Staubli VAL3: HIT_YD.pjx

--- HIT_YD.pjx ---
Parameters version=s7.6.4 stackSize=5000 millimeterUnit=true
Program file=blow.pgx
Program file=bypassPick.pgx
Program file=cellManager.pgx
Program file=getToolStatus.pgx
Program file=goHome.pgx
Program file=init.pgx
Program file=initTracking.pgx
Program file=isInSafetyArea.pgx
Program file=ModbusGet.pgx
Program file=modbusSet.pgx
Program file=OMAC_Abort.pgx
Program file=OMAC_Hold.pgx
Program file=OMAC_Main.pgx
Program file=OMAC_Reset.pgx
Program file=OMAC_Start.pgx
Program file=OMAC_Stop.pgx
Program file=OMAC_Unhold.pgx
Program file=overflowPick.pgx
Program file=Place.pgx
Program file=productionCycle.pgx
Program file=robot2PC.pgx
Program file=robot2PLC.pgx
Program file=send2NextRob.pgx
Program file=setAlarm.pgx
Program file=setConvSpeed.pgx
Program file=start.pgx
Program file=stop.pgx
Program file=trackErr_init.pgx
Program file=trackingPick.pgx
Program file=transferQueue.pgx
Data file=HIT_YD.dtx
Library alias=mot path=Disk://Tracking/Motion/Motion.pjx
Type name=object path=Disk://Tracking/Templates/object/object.pjx

--- HIT_YD.dtx ---
aio aConvSpeed = {link=ModbusSrv-0\Modbus-Word\ao[3]}
aio aPlcCmd = {link=ModbusSrv-0\Modbus-Word\ai[0]}
aio aRbAlarm = {link=ModbusSrv-0\Modbus-Word\ao[0]}
aio aRbStatus = {link=ModbusSrv-0\Modbus-Word\ao[1]}
bool _bConvExist = true
bool _bEndCycle
bool _bIsPicking
bool _bIsPlacing
bool _bMutexCnvQueue
bool _bOverflowed = true
bool _bPartInTool = true
bool _bSentToHome
bool _bVisionOK = true
bool bLockPage
bool bPickDetection
bool bSetConvSpeed
bool bSyn
bool bTransferData = true
dio dAlarm[8]
  [0] = {link=ModbusSrv-0\Modbus-Bit\do[8]}
  [1] = {link=ModbusSrv-0\Modbus-Bit\do[9]}
  [2] = {link=ModbusSrv-0\Modbus-Bit\do[10]}
  [3] = {link=ModbusSrv-0\Modbus-Bit\do[11]}
  [4] = {link=ModbusSrv-0\Modbus-Bit\do[12]}
  [5] = {link=ModbusSrv-0\Modbus-Bit\do[13]}
  [6] = {link=ModbusSrv-0\Modbus-Bit\do[14]}
  [7] = {link=ModbusSrv-0\Modbus-Bit\do[15]}
dio dBlow = {link=BasicIO-1\%Q5}
dio dConvControl[2]
  [0] = {link=BasicIO-1\%I4}
  [1] = {link=BasicIO-1\%Q6}
dio dPartInTool = {link=fIn0}
dio dPermitPlace[4]
  [0] = {link=BasicIO-1\%I3}
  [1] = {link=BasicIO-1\%I2}
  [2] = {link=BasicIO-1\%I1}
  [3] = {link=BasicIO-1\%I0}
dio dPlaceDone[4]
  [0] = {link=BasicIO-1\%Q11}
  [1] = {link=BasicIO-1\%Q10}
  [2] = {link=BasicIO-1\%Q9}
  [3] = {link=BasicIO-1\%Q8}
dio dStartControl[4]
  [0] = {link=ModbusSrv-0\Modbus-Bit\di[4]}
  [1] = {link=ModbusSrv-0\Modbus-Bit\di[5]}
  [2] = {link=ModbusSrv-0\Modbus-Bit\di[6]}
  [3] = {link=ModbusSrv-0\Modbus-Bit\di[7]}
dio dStartState[4]
  [0] = {link=ModbusSrv-0\Modbus-Bit\do[4]}
  [1] = {link=ModbusSrv-0\Modbus-Bit\do[5]}
  [2] = {link=ModbusSrv-0\Modbus-Bit\do[6]}
  [3] = {link=ModbusSrv-0\Modbus-Bit\do[7]}
dio dVacuum = {link=BasicIO-1\%Q4}
frame fConveyor = {x=365.904087, y=326.91934, z=-82.602337, rx=-0.010861, ry=-0.059106, rz=0.004608, fatherId=world[0]}
frame fDetection = {x=392.598601, y=461.346273, z=-82.976862, rx=0.205045, ry=0.617271, rz=0.011036, fatherId=world[0]}
jointRs jDropPart = {j1=102.785955, j2=-95.43121, j3=69.578977, j4=134.260732}
jointRs jHome = {j1=102.785955, j2=-95.43121, j3=69.578977, j4=134.260732}
jointRs jPark = {j1=102.785955, j2=-95.43121, j3=69.578977, j4=134.260732}
mdesc _mLoad = {accel=133.4025, vel=115.5, decel=133.4025}
mdesc mLoad = {accel=121, vel=110, decel=121}
mdesc mNomSpeed = {accel=144, vel=120, decel=144, leave=20, reach=20}
mdesc mPickDown = {accel=144, vel=120, decel=144, leave=10, reach=10, blend=off}
mdesc mPickup = {accel=121, vel=110, decel=121, leave=40, reach=40}
mdesc mPlaceDown = {accel=144, vel=120, decel=144, leave=15, reach=15, blend=off}
mdesc mPlaceUp = {accel=144, vel=120, decel=144, leave=20, reach=20, blend=cartesian}
mdesc mSlow = {accel=1, vel=10, decel=1, leave=10, reach=10}
mdesc mUnload = {accel=144, vel=120, decel=144, leave=40, reach=40}
num _nBlowDelay
num _nCntBypassed = 1
num _nCntPartsDone[2]
  [0] = 74956
  [1] = 74907
num _nCntTransfered = 8
num _nConvSpd
num _nCycleTime[4]
  [0] = 33.16
  [1] = 2.331
  [2] = 48.87
  [3] = 0.935
num _nCycleTimeIndx
num _nID = -1
num _nLastStateCMD
num _nOmacStat = 3
num _nPartID = 1
num _nPlaceCurItem[2]
num _nPullIndexTQ = 8
num _nPushIndexTQ = 8
num _nStateCMD
num _nTimer = 355.546
num _nTrackErr = 315
num nBlowID = 0.3
num nBypass = 1
num nLoadRatio[4]
  [0] = 0.7
  [1] = 0.85
  [2] = 0.95
  [3] = 1.05
num nNomConvSpeed = 100
num nPartHeight = 6
num nPickAppro = 65
num nPickOS_X = -3
num nPickOS_Y
num nPlaceAppro = 60
public num nPlaceNum = 3
num nSafeMaxX = 850
num nSafeMaxY = 650
num nSafeMinX
num nSafeMinY
num nStopTime = 0.02
num nTestData[5]
  [0] = 6
  [1] = -49
  [2] = 55
  [4] = 24206
num nVacuumID
num nWaitDist2Up4BP = -300
num nWaitDistToDown = 50
num nWaitDistToUp[1 3]
  [0,0] = -80
  [0,1] = 120
  [0,2] = 400
num nWaitDistX
object _oTransferQueue[1 100]
  [0,0]
    num nID = -1
    num nLatchedValue
    trsf trTrsf
  [0,1]
    num nID = -1
    num nLatchedValue
    trsf trTrsf
  [0,2]
    num nID = -1
    num nLatchedValue
    trsf trTrsf
  [0,3]
    num nID = -1
    num nLatchedValue
    trsf trTrsf
  [0,4]
    num nID = -1
    num nLatchedValue
    trsf trTrsf
  [0,5]
    num nID = -1
    num nLatchedValue
    trsf trTrsf
  [0,6]
    num nID = -1
    num nLatchedValue
    trsf trTrsf
  [0,7]
    num nID = -1
    num nLatchedValue
    trsf trTrsf
  [0,8]
    num nID = -1
    num nLatchedValue
    trsf trTrsf
  [0,9]
    num nID = -1
    num nLatchedValue
    trsf trTrsf
  [0,10]
    num nID = -1
    num nLatchedValue
    trsf trTrsf
  [0,11]
    num nID = -1
    num nLatchedValue
    trsf trTrsf
  [0,12]
    num nID = -1
    num nLatchedValue
    trsf trTrsf
  [0,13]
    num nID = -1
    num nLatchedValue
    trsf trTrsf
  [0,14]
    num nID = -1
    num nLatchedValue
    trsf trTrsf
  [0,15]
    num nID = -1
    num nLatchedValue
    trsf trTrsf
  [0,16]
    num nID = -1
    num nLatchedValue
    trsf trTrsf
  [0,17]
    num nID = -1
    num nLatchedValue
    trsf trTrsf
  [0,18]
    num nID = -1
    num nLatchedValue
    trsf trTrsf
  [0,19]
    num nID = -1
    num nLatchedValue
    trsf trTrsf
  [0,20]
    num nID = -1
    num nLatchedValue
    trsf trTrsf
  [0,21]
    num nID = -1
    num nLatchedValue
    trsf trTrsf
  [0,22]
    num nID = -1
    num nLatchedValue
    trsf trTrsf
  [0,23]
    num nID = -1
    num nLatchedValue
    trsf trTrsf
  [0,24]
    num nID = -1
    num nLatchedValue
    trsf trTrsf
  [0,25]
    num nID = -1
    num nLatchedValue
    trsf trTrsf
  [0,26]
    num nID = -1
    num nLatchedValue
    trsf trTrsf
  [0,27]
    num nID = -1
    num nLatchedValue
    trsf trTrsf
  [0,28]
    num nID = -1
    num nLatchedValue
    trsf trTrsf
  [0,29]
    num nID = -1
    num nLatchedValue
    trsf trTrsf
  [0,30]
    num nID = -1
    num nLatchedValue
    trsf trTrsf
  [0,31]
    num nID = -1
    num nLatchedValue
    trsf trTrsf
  [0,32]
    num nID = -1
    num nLatchedValue
    trsf trTrsf
  [0,33]
    num nID = -1
    num nLatchedValue
    trsf trTrsf
  [0,34]
    num nID = -1
    num nLatchedValue
    trsf trTrsf
  [0,35]
    num nID = -1
    num nLatchedValue
    trsf trTrsf
  [0,36]
    num nID = -1
    num nLatchedValue
    trsf trTrsf
  [0,37]
    num nID = -1
    num nLatchedValue
    trsf trTrsf
  [0,38]
    num nID = -1
    num nLatchedValue
    trsf trTrsf
  [0,39]
    num nID = -1
    num nLatchedValue
    trsf trTrsf
  [0,40]
    num nID = -1
    num nLatchedValue
    trsf trTrsf
  [0,41]
    num nID = -1
    num nLatchedValue
    trsf trTrsf
  [0,42]
    num nID = -1
    num nLatchedValue
    trsf trTrsf
  [0,43]
    num nID = -1
    num nLatchedValue
    trsf trTrsf
  [0,44]
    num nID = -1
    num nLatchedValue
    trsf trTrsf
  [0,45]
    num nID = -1
    num nLatchedValue
    trsf trTrsf
  [0,46]
    num nID = -1
    num nLatchedValue
    trsf trTrsf
  [0,47]
    num nID = -1
    num nLatchedValue
    trsf trTrsf
  [0,48]
    num nID = -1
    num nLatchedValue
    trsf trTrsf
  [0,49]
    num nID = -1
    num nLatchedValue
    trsf trTrsf
  [0,50]
    num nID = -1
    num nLatchedValue
    trsf trTrsf
  [0,51]
    num nID = -1
    num nLatchedValue
    trsf trTrsf
  [0,52]
    num nID = -1
    num nLatchedValue
    trsf trTrsf
  [0,53]
    num nID = -1
    num nLatchedValue
    trsf trTrsf
  [0,54]
    num nID = -1
    num nLatchedValue
    trsf trTrsf
  [0,55]
    num nID = -1
    num nLatchedValue
    trsf trTrsf
  [0,56]
    num nID = -1
    num nLatchedValue
    trsf trTrsf
  [0,57]
    num nID = -1
    num nLatchedValue
    trsf trTrsf
  [0,58]
    num nID = -1
    num nLatchedValue
    trsf trTrsf
  [0,59]
    num nID = -1
    num nLatchedValue
    trsf trTrsf
  [0,60]
    num nID = -1
    num nLatchedValue
    trsf trTrsf
  [0,61]
    num nID = -1
    num nLatchedValue
    trsf trTrsf
  [0,62]
    num nID = -1
    num nLatchedValue
    trsf trTrsf
  [0,63]
    num nID = -1
    num nLatchedValue
    trsf trTrsf
  [0,64]
    num nID = -1
    num nLatchedValue
    trsf trTrsf
  [0,65]
    num nID = -1
    num nLatchedValue
    trsf trTrsf
  [0,66]
    num nID = -1
    num nLatchedValue
    trsf trTrsf
  [0,67]
    num nID = -1
    num nLatchedValue
    trsf trTrsf
  [0,68]
    num nID = -1
    num nLatchedValue
    trsf trTrsf
  [0,69]
    num nID = -1
    num nLatchedValue
    trsf trTrsf
  [0,70]
    num nID = -1
    num nLatchedValue
    trsf trTrsf
  [0,71]
    num nID = -1
    num nLatchedValue
    trsf trTrsf
  [0,72]
    num nID = -1
    num nLatchedValue
    trsf trTrsf
  [0,73]
    num nID = -1
    num nLatchedValue
    trsf trTrsf
  [0,74]
    num nID = -1
    num nLatchedValue
    trsf trTrsf
  [0,75]
    num nID = -1
    num nLatchedValue
    trsf trTrsf
  [0,76]
    num nID = -1
    num nLatchedValue
    trsf trTrsf
  [0,77]
    num nID = -1
    num nLatchedValue
    trsf trTrsf
  [0,78]
    num nID = -1
    num nLatchedValue
    trsf trTrsf
  [0,79]
    num nID = -1
    num nLatchedValue
    trsf trTrsf
  [0,80]
    num nID = -1
    num nLatchedValue
    trsf trTrsf
  [0,81]
    num nID = -1
    num nLatchedValue
    trsf trTrsf
  [0,82]
    num nID = -1
    num nLatchedValue
    trsf trTrsf
  [0,83]
    num nID = -1
    num nLatchedValue
    trsf trTrsf
  [0,84]
    num nID = -1
    num nLatchedValue
    trsf trTrsf
  [0,85]
    num nID = -1
    num nLatchedValue
    trsf trTrsf
  [0,86]
    num nID = -1
    num nLatchedValue
    trsf trTrsf
  [0,87]
    num nID = -1
    num nLatchedValue
    trsf trTrsf
  [0,88]
    num nID = -1
    num nLatchedValue
    trsf trTrsf
  [0,89]
    num nID = -1
    num nLatchedValue
    trsf trTrsf
  [0,90]
    num nID = -1
    num nLatchedValue
    trsf trTrsf
  [0,91]
    num nID = -1
    num nLatchedValue
    trsf trTrsf
  [0,92]
    num nID = -1
    num nLatchedValue
    trsf trTrsf
  [0,93]
    num nID = -1
    num nLatchedValue
    trsf trTrsf
  [0,94]
    num nID = -1
    num nLatchedValue
    trsf trTrsf
  [0,95]
    num nID = -1
    num nLatchedValue
    trsf trTrsf
  [0,96]
    num nID = -1
    num nLatchedValue
    trsf trTrsf
  [0,97]
    num nID = -1
    num nLatchedValue
    trsf trTrsf
  [0,98]
    num nID = -1
    num nLatchedValue
    trsf trTrsf
  [0,99]
    num nID = -1
    num nLatchedValue
    trsf trTrsf
pointRs pPick = {shoulder=lefty, fatherId=fDetection[0]}
pointRs pPlace[4]
  [0] = {x=356.46, y=115, z=-70.81, rx=180, rz=-98.019983, shoulder=lefty, fatherId=world[0]}
  [1] = {x=486.131736, y=115, z=-70.81, rx=180, rz=-98.021161, shoulder=lefty, fatherId=world[0]}
  [2] = {x=630, y=105, z=-70.81, rx=180, rz=-98.02183, shoulder=lefty, fatherId=world[0]}
  [3] = {x=770, y=105, z=-70.8, rx=180, rz=-98.02084, shoulder=lefty, fatherId=world[0]}
sio skToRobot = {link=Socket\toRobot_sk1}
sio sktoPC = {link=Socket\toPC}
sio synServer = {link=Socket\synRobot1}
string _sCycleStatus = "Distance to pick:  -79.66"
string sConveyorList = "cvIn"
string sDataPC = "stop"
string sString = "done"
tool tGripper = {z=85, rz=45, fatherId=flange[0], ioLink=valve1}

--- initTracking.pgx ---
program initTracking()
  local num l_nConvNum
  local num l_nError
  local string l_sErrorMessage
begin
  // This program initializes all tracking variables and launches all tracking tasks
  //
  // Input parameters
  //  None            :
  //
  // Output parameters
  //  None            :
  //
  //----------------------------------------------------------------
  //
  // Load motion library
  l_nError=mot:libLoad("Tracking\Motion")
  if l_nError!=0
    popUpMsg("Error while loading motion library: "+toString("",l_nError))
  endIf
  //
  // Start the libraries to perform conveyor tracking
  call mot:create(sConveyorList)
  //
  // Waits until all tasks are up and running
  for l_nConvNum=0 to size(sConveyorList)-1
    do
      call mot:getStatus(l_nConvNum,l_nError)
      delay(0)
    until (l_nError==0)
  endFor
  _bConvExist=true
  //
  //Reads the position of the frames defined with the Wizard,
  //for all conveyors on the conveyor list
  for l_nConvNum=0 to size(sConveyorList)-1
    // Get the conveyor frame
    call mot:getConvFrame(l_nConvNum,fConveyor[l_nConvNum],world,l_nError)
    if l_nError!=0
      call mot:getErrorMessage(l_sErrorMessage)
      popUpMsg(l_sErrorMessage)
    endIf
    //
    // Get the detection frame
    call mot:getDetectFrame(l_nConvNum,fDetection[l_nConvNum],world,l_nError)
    if l_nError!=0
      call mot:getErrorMessage(l_sErrorMessage)
      popUpMsg(l_sErrorMessage)
    endIf
  endFor
  //
end

--- isInSafetyArea.pgx ---
program isInSafetyArea()
  local jointRs l_jHere
  local num l_ns
  local pointRs l_pCurrent
begin
  do
    l_pCurrent=here(flange,world)
    //**************************************************//
    //******** 用来判断机器人是否在安全工作空间 ********//
    //**************************************************//
    if (l_pCurrent.trsf.y>=nSafeMaxY or l_pCurrent.trsf.y<=nSafeMinY or l_pCurrent.trsf.x>=nSafeMaxX or l_pCurrent.trsf.x<=nSafeMinX) and _nOmacStat==3
      aioSet(aRbAlarm,10)
      call setAlarm(7)
      popUpMsg("机器人超出安全工作空间！")
      logMsg("机器人超出安全工作空间！")
      call OMAC_Abort()
    endIf

    if (dConvControl[0]==true)
      dConvControl[1]=true
    else
      dConvControl[1]=false
    endIf
    delay(0)
  until false
end

--- OMAC_Reset.pgx ---
program OMAC_Reset()
  local bool l_bResult
  local joint l_jHere
  local num l_nKey
begin

  //OMAC进程:resetting
  _nOmacStat=4
  logMsg("上位机手动操作：复位")



  // Reset conveyor speed
  //  call setConvSpeed(0,0)
  //start vision
  _bVisionOK=false
  if taskStatus("robot2PC")>=0
    taskKill("robot2PC")
  endIf
  wait(taskStatus("robot2PC")<0)
  taskCreate "robot2PC",100,robot2PC()
  //wait vision ok
  l_bResult=watch(_bVisionOK,5)
  if l_bResult==false
    //alarm
    call setAlarm(0)
    logMsg("vision start failed")
    taskKill("robot2PC")
    _nOmacStat=9
    return
  endIf
  // Variable initializing
  call init()
  call trackErr_init()
  // Launch Tracking
  call initTracking()
  if !isInRange(herej())
    aioSet(aRbAlarm,20)
    call setAlarm(1)
    popUpMsg("机器人关节超限!")
    taskCreate "Abort",100,OMAC_Abort()
    return
  endIf
  //
  resetMotion()
  // Enables arm power
  while !isPowered()
    enablePower()
    delay(1)
  endWhile
  _bSentToHome=true
  // Send robot to home position
  l_jHere=herej()
  l_jHere.j3=jHome.j3
  movej(l_jHere,tGripper,mSlow)
  movej(jHome,tGripper,mSlow)
  //
  //
  // Init user screen
  cls()
  gotoxy(0,4)
  put("Cycle Time (Last):    ")
  gotoxy(0,6)
  put("Cycle Time (Average): ")
  gotoxy(0,8)
  put("Cycle Time (Best):    ")
  gotoxy(0,10)
  put("      Pick                Place         ")
  gotoxy(0,11)
  put("  Done   Transfer      Done   ")


  //Launch queue transfer tasks
  if bTransferData[0]
    if taskStatus("TransferQueue1")>=0
      taskKill("TransferQueue1")
    endIf
    taskCreate "TransferQueue1",100,transferQueue(0)
    wait(taskStatus("TransferQueue1")==1)
  endIf

  // Task to remove picking positions that have pass the downstream limit while the robot is placing a part.
  if taskStatus("overflowPick")>=0
    taskKill("overflowPick")
  endIf
  taskCreate "overflowPick",100,overflowPick()
  wait(taskStatus("overflowPick")==1)

  //OMAC进程:ready
  _nOmacStat=1
  delay(0)
end

--- overflowPick.pgx ---
program overflowPick()
  local num l_nConvNum
  local num l_nConvSpeed
  local num l_nConvSpeedOld
  local num l_nDistDown
  local num l_nDistUp
  local num l_nEncLatchVal
  local num l_nError
  local num l_nLimCrossPer
begin
  // This program removes all the objects from the conveyor’s queue
  //  that the robot is not going to work with. It removes the
  //  objects by overflow or by bypass.
  // The use of this program on a task allows to remove the
  //  unnecessary objects from the conveyor’s queue while the robot
  //  is working with a previous object.
  // If the variable bTransferData is set to true, the program will
  //  send the objects to the transfer queue before removing the
  //  objects from the conveyor’s queue.
  // If the variable bSetConvSpeed is set to true, the program will
  //  reduce/stop the conveyor to avoid that an object leaves the
  //  tracking window.
  //
  // Input parameters
  //  None            :
  //
  // Output parameters
  //  None            :
  //
  //----------------------------------------------------------------
  //
  l_nConvNum=0
  l_nConvSpeed=0
  l_nConvSpeedOld=0
  //
  do
    //
    // Takes control of the Pick conveyor queue
    setMutex(_bMutexCnvQueue[l_nConvNum])
    //
    // Remove objects by Bypass
    if nBypass[l_nConvNum]>0 and _nCntBypassed[l_nConvNum]==0
      if _bOverflowed and false
        _bOverflowed=false
        _nCntBypassed=nBypass
      else
        call bypassPick()
      endIf
      //call bypassPick()
    endIf
    //
    // Check if there is an object on the conveyor’s queue
    if _nID[l_nConvNum]==-1
      call mot:getNextID(l_nConvNum,_nID[l_nConvNum])
    endIf
    //
    // If there is an object on the conveyor’s queue: Remove the object from the conveyor’s
    //  queue if the object has passed the downstream limit (overflow) or, if the variable
    //  setConvSpeed is set to true, stop the conveyor before the object crosses the downstream limit.
    if _nID[l_nConvNum]!=-1
      // Recover next object transformation from the stack
      call mot:getObjectData(l_nConvNum,pPick.trsf,l_nError)
      call mot:getDistance(l_nConvNum,pPick,0,l_nDistUp,l_nDistDown,l_nError)
      // Reduce/stop the speed of the conveyor when the object is in between the two middle limits.
      //  The value of the speed is calculated as a percentage of the nominal speed. The percentage
      //  is proportional to the distance of the object to the middle limits, 100% when the object
      //  is at the first middle limit and 0% when the object is at the second middle limit.
      if bSetConvSpeed[l_nConvNum] and l_nDistDown<nWaitDistToDown[l_nConvNum]
        l_nLimCrossPer=max((nWaitDistToUp[l_nConvNum,2]-l_nDistUp)/(nWaitDistToUp[l_nConvNum,2]-nWaitDistToUp[l_nConvNum,1]),0)
        l_nConvSpeed=l_nLimCrossPer*nNomConvSpeed[l_nConvNum]
        if l_nConvSpeedOld!=l_nConvSpeed
          call setConvSpeed(l_nConvNum,sel(l_nDistUp>nWaitDistToUp[l_nConvNum,1],l_nConvSpeed,nNomConvSpeed[l_nConvNum]))
          l_nConvSpeedOld=l_nConvSpeed
        endIf
      else
        // Remove objects by Overflow
        if (l_nDistUp>nWaitDistToUp[l_nConvNum,1])
          //
          // Send object to the next robot
          if bTransferData[l_nConvNum]
            call mot:getObjectLatch(l_nConvNum,l_nEncLatchVal,l_nError)
            call send2NextRob(l_nConvNum,_nID[l_nConvNum],pPick.trsf,l_nEncLatchVal)
          endIf
          //
          // Remove object from conveyor's queue
          call mot:removePart(l_nConvNum)
          _nID[l_nConvNum]=-1
          pPick.trsf={0,0,0,0,0,0}
          _bOverflowed=true
          _nCntTransfered[l_nConvNum]=_nCntTransfered[l_nConvNum]+1
        endIf
      endIf
    else
      // No object available => full speed on the conveyor
      l_nConvSpeed=nNomConvSpeed[l_nConvNum]
      if bSetConvSpeed[l_nConvNum] and l_nConvSpeedOld!=l_nConvSpeed
        call setConvSpeed(l_nConvNum,l_nConvSpeed)
        l_nConvSpeedOld=l_nConvSpeed
      endIf
    endIf
    //
    // Release control of the Pick conveyor queue.
    _bMutexCnvQueue[l_nConvNum]=false
    //
    delay(0)
  until false
end

--- productionCycle.pgx ---
program productionCycle()
  local bool l_bPartDone
  local num l_nNum
  local string l_sToolStatus
begin
  // This program is the main cycle. It pick on part from the input
  // conveyor and places it on an empty cavity on the output conveyor.
  //
  // Input parameters
  //  None            :
  //
  // Output parameters
  //  None            :
  //
  //----------------------------------------------------------------
  //
  // In order to improve cycle time, vacuum is always on, even while
  //  placing a part. To place a part, the blow is activated for a
  //  short period of time when the robot arrives to the place position.
  //
  // Main loop

  //---------------------------------------------------------------------//
  //call ServerGet(sFirstRStatus)
  do
    //Takes control of the Pick conveyor queue.
    setMutex(_bMutexCnvQueue[0])
    do
      call trackingPick(l_bPartDone)
      delay(0)
    until l_bPartDone
    // Release control of the Pick conveyor queue.
    _bMutexCnvQueue[0]=false

    //
    call place()
    //
    delay(0)
  until _bEndCycle
  _bEndCycle=true
  //
end

--- robot2PC.pgx ---
program robot2PC()
begin

  clearBuffer(sktoPC)
  sktoPC="run"
  sDataPC=sktoPC
  _bVisionOK=true
end

--- setAlarm.pgx ---
program setAlarm(num x_nNum)
  local num l_ns
begin
  switch x_nNum
    case 0
      dAlarm[0]=true
      dAlarm[1]=false
      dAlarm[2]=false
      dAlarm[3]=false
      dAlarm[4]=false
      dAlarm[5]=false
      dAlarm[6]=false
      dAlarm[7]=false
      delay(0.35)
      dAlarm[0]=false
      dAlarm[1]=false
      dAlarm[2]=false
      dAlarm[3]=false
      dAlarm[4]=false
      dAlarm[5]=false
      dAlarm[6]=false
      dAlarm[7]=false
    break
    case 1
      dAlarm[0]=false
      dAlarm[1]=true
      dAlarm[2]=false
      dAlarm[3]=false
      dAlarm[4]=false
      dAlarm[5]=false
      dAlarm[6]=false
      dAlarm[7]=false
      delay(0.35)
      dAlarm[0]=false
      dAlarm[1]=false
      dAlarm[2]=false
      dAlarm[3]=false
      dAlarm[4]=false
      dAlarm[5]=false
      dAlarm[6]=false
      dAlarm[7]=false
    break
    case 2
      dAlarm[0]=false
      dAlarm[1]=false
      dAlarm[2]=true
      dAlarm[3]=false
      dAlarm[4]=false
      dAlarm[5]=false
      dAlarm[6]=false
      dAlarm[7]=false
      delay(0.35)
      dAlarm[0]=false
      dAlarm[1]=false
      dAlarm[2]=false
      dAlarm[3]=false
      dAlarm[4]=false
      dAlarm[5]=false
      dAlarm[6]=false
      dAlarm[7]=false
    break
    case 3
      dAlarm[0]=false
      dAlarm[1]=false
      dAlarm[2]=true
      dAlarm[3]=false
      dAlarm[4]=false
      dAlarm[5]=false
      dAlarm[6]=false
      dAlarm[7]=false
      delay(0.35)
      dAlarm[0]=false
      dAlarm[1]=false
      dAlarm[2]=false
      dAlarm[3]=false
      dAlarm[4]=false
      dAlarm[5]=false
      dAlarm[6]=false
      dAlarm[7]=false
    break
    case 4
      dAlarm[0]=false
      dAlarm[1]=false
      dAlarm[2]=false
      dAlarm[3]=false
      dAlarm[4]=true
      dAlarm[5]=false
      dAlarm[6]=false
      dAlarm[7]=false
      delay(0.35)
      dAlarm[0]=false
      dAlarm[1]=false
      dAlarm[2]=false
      dAlarm[3]=false
      dAlarm[4]=false
      dAlarm[5]=false
      dAlarm[6]=false
      dAlarm[7]=false
    break
    case 5
      dAlarm[0]=false
      dAlarm[1]=false
      dAlarm[2]=false
      dAlarm[3]=false
      dAlarm[4]=false
      dAlarm[5]=true
      dAlarm[6]=false
      dAlarm[7]=false
      delay(0.35)
      dAlarm[0]=false
      dAlarm[1]=false
      dAlarm[2]=false
      dAlarm[3]=false
      dAlarm[4]=false
      dAlarm[5]=false
      dAlarm[6]=false
      dAlarm[7]=false
    break
    case 6
      dAlarm[0]=false
      dAlarm[1]=false
      dAlarm[2]=false
      dAlarm[3]=false
      dAlarm[4]=false
      dAlarm[5]=false
      dAlarm[6]=true
      dAlarm[7]=false
      delay(0.35)
      dAlarm[0]=false
      dAlarm[1]=false
      dAlarm[2]=false
      dAlarm[3]=false
      dAlarm[4]=false
      dAlarm[5]=false
      dAlarm[6]=false
      dAlarm[7]=false
    break
    case 7
      dAlarm[0]=false
      dAlarm[1]=false
      dAlarm[2]=false
      dAlarm[3]=false
      dAlarm[4]=false
      dAlarm[5]=false
      dAlarm[6]=false
      dAlarm[7]=true
      delay(0.35)
      dAlarm[0]=false
      dAlarm[1]=false
      dAlarm[2]=false
      dAlarm[3]=false
      dAlarm[4]=false
      dAlarm[5]=false
      dAlarm[6]=false
      dAlarm[7]=false
    break
    default
      dAlarm[0]=false
      dAlarm[1]=false
      dAlarm[2]=false
      dAlarm[3]=false
      dAlarm[4]=false
      dAlarm[5]=false
      dAlarm[6]=false
      dAlarm[7]=false
    break
  endSwitch
end

--- transferQueue.pgx ---
program transferQueue(num x_nConvNum (dimensions=1))
  local num l_nError
begin
  // This program sends to the next robot the objects presents on
  //  the transfer queue.
  //
  // Input parameters
  //  x_nConvNum      : Conveyor number
  //
  // Output parameters
  //  None            :
  //
  //----------------------------------------------------------------
  //
  clearBuffer(skToRobot[x_nConvNum])
  do
    // If the ID of the next element of the queue is greater than -1,
    //  it means that the element contains the information of an object,
    //  therefore it has to be sent to the next robot.
    if _oTransferQueue[x_nConvNum,_nPullIndexTQ[x_nConvNum]].nID>-1
      // Send the object to the next robot
      call mot:sendToNextRobot(skToRobot[x_nConvNum],0,_oTransferQueue[x_nConvNum,_nPullIndexTQ[x_nConvNum]].nID,_oTransferQueue[x_nConvNum,_nPullIndexTQ[x_nConvNum]].trTrsf,_oTransferQueue[x_nConvNum,_nPullIndexTQ[x_nConvNum]].nLatchedValue,l_nError)
      if l_nError>0
        popUpMsg("Part not sent, error code over skToRobot["+toString("",x_nConvNum)+"]: "+toString("",l_nError))
      endIf
      // Erase the object from the queue.
      _oTransferQueue[x_nConvNum,_nPullIndexTQ[x_nConvNum]].nLatchedValue=0
      _oTransferQueue[x_nConvNum,_nPullIndexTQ[x_nConvNum]].trTrsf={0,0,0,0,0,0}
      // The last value erased is the ID. The program send2NextRob is looking to
      //  this value in order to know if the element of the queue is free.
      _oTransferQueue[x_nConvNum,_nPullIndexTQ[x_nConvNum]].nID=-1
      _nPullIndexTQ[x_nConvNum]=(_nPullIndexTQ[x_nConvNum]+1)%size(_oTransferQueue,2)
    endIf
    delay(0)
  until false
end
